TYPE PT1T2_Parameter_Strukt :
STRUCT
	K :			REAL;
	T1 :		REAL;
	T2 :		REAL;
END_STRUCT
END_TYPE

(* stored: Version 1.1.0.1, ProductVersion 3.1.4024.13
   DUT PT1T2_Parameter_Strukt: Id {23a5cb93-4cf2-48d5-b112-3b6fa044df40} *)
